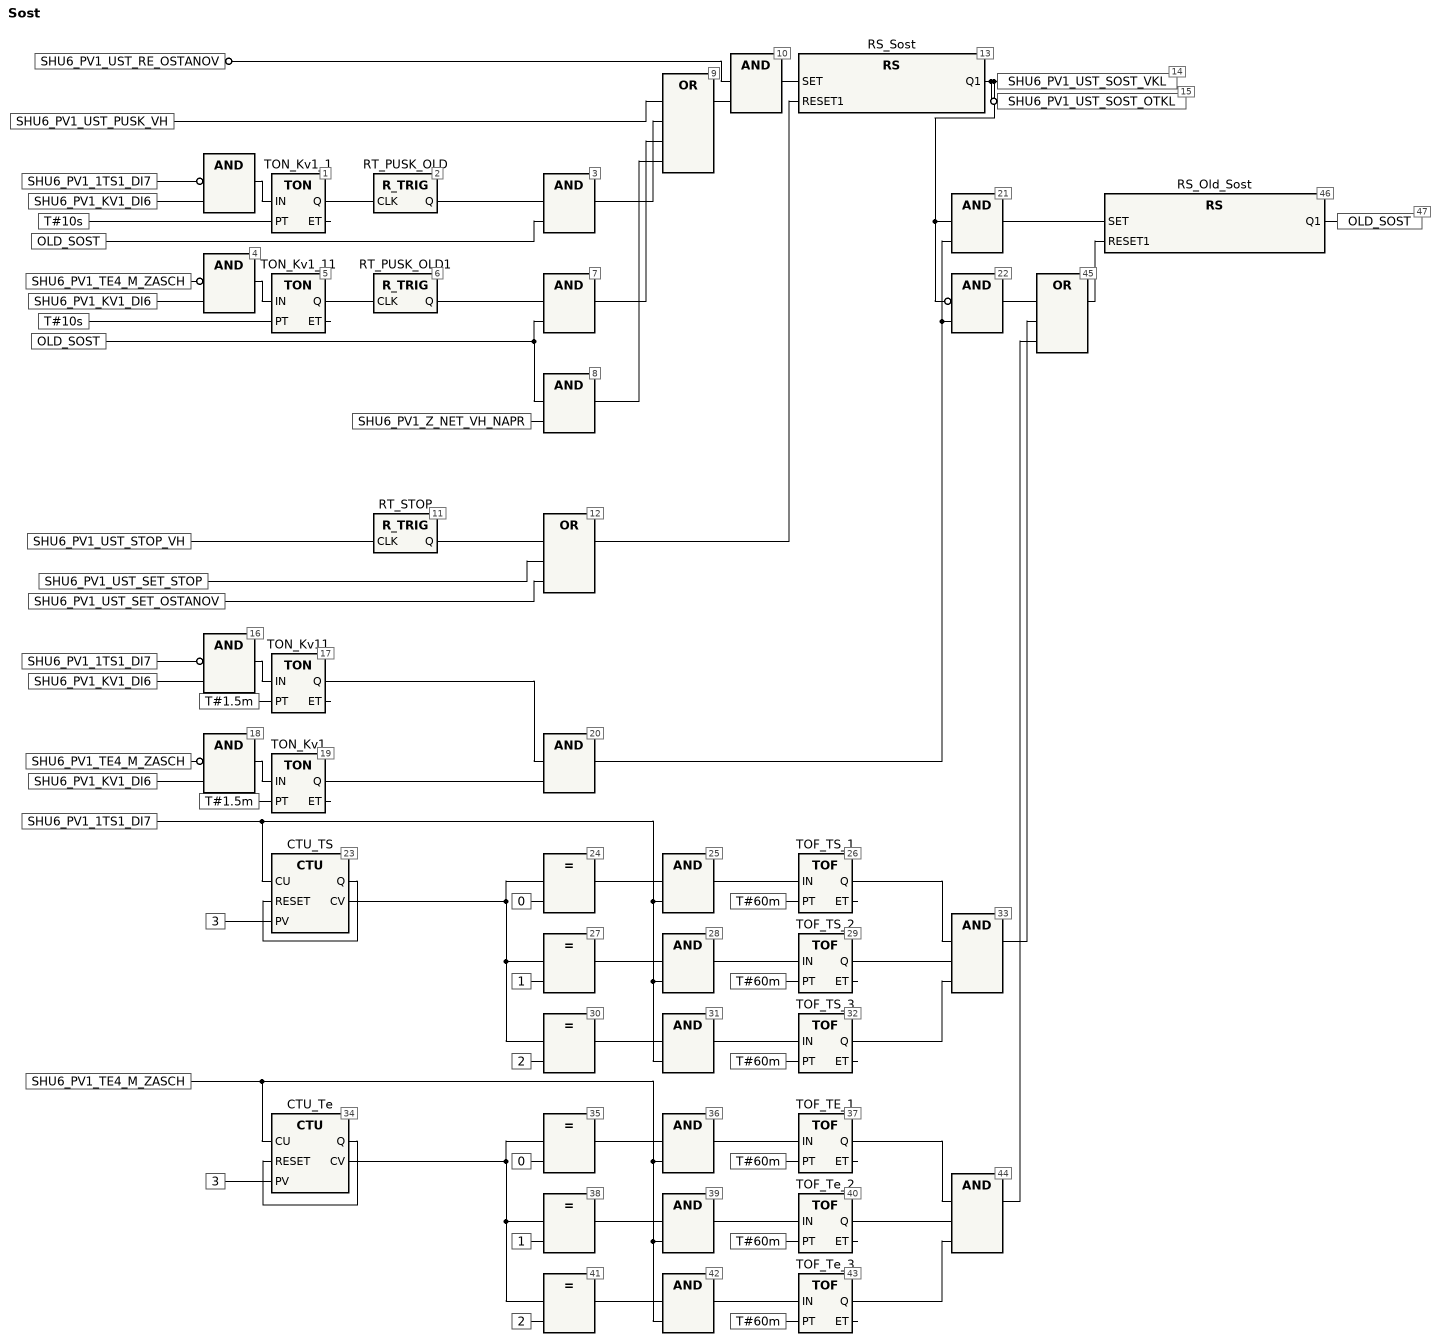
_CFC_ (* Continuous Function Chart, elements in execution order *)
#0 AND(NOT SHU6_PV1_1TS1_DI7, SHU6_PV1_KV1_DI6)
#1 TON_Kv1_1:TON(IN: #0, PT: T#10s)
#2 RT_PUSK_OLD:R_TRIG(CLK: #1.Q)
#3 AND(#2.Q, OLD_SOST)
#4 AND(NOT SHU6_PV1_TE4_M_ZASCH, SHU6_PV1_KV1_DI6)
#5 TON_Kv1_11:TON(IN: #4, PT: T#10s)
#6 RT_PUSK_OLD1:R_TRIG(CLK: #5.Q)
#7 AND(#6.Q, OLD_SOST)
#8 AND(OLD_SOST, SHU6_PV1_Z_NET_VH_NAPR)
#9 OR(SHU6_PV1_UST_PUSK_VH, #3, #7, #8)
#10 AND(NOT SHU6_PV1_UST_RE_OSTANOV, #9)
#11 RT_STOP:R_TRIG(CLK: SHU6_PV1_UST_STOP_VH)
#12 OR(#11.Q, SHU6_PV1_UST_SET_STOP, SHU6_PV1_UST_SET_OSTANOV)
#13 RS_Sost:RS(SET: #10, RESET1: #12)
#14 SHU6_PV1_UST_SOST_VKL <= #13.Q1
#15 SHU6_PV1_UST_SOST_OTKL <= NOT #13.Q1
#16 AND(NOT SHU6_PV1_1TS1_DI7, SHU6_PV1_KV1_DI6)
#17 TON_Kv11:TON(IN: #16, PT: T#1.5m)
#18 AND(NOT SHU6_PV1_TE4_M_ZASCH, SHU6_PV1_KV1_DI6)
#19 TON_Kv1:TON(IN: #18, PT: T#1.5m)
#20 AND(#17.Q, #19.Q)
#21 AND(#13.Q1, #20)
#22 AND(NOT #13.Q1, #20)
#23 CTU_TS:CTU(CU: SHU6_PV1_1TS1_DI7, RESET: #23.Q, PV: 3)
#24 =(#23.CV, 0)
#25 AND(#24, SHU6_PV1_1TS1_DI7)
#26 TOF_TS_1:TOF(IN: #25, PT: T#60m)
#27 =(#23.CV, 1)
#28 AND(#27, SHU6_PV1_1TS1_DI7)
#29 TOF_TS_2:TOF(IN: #28, PT: T#60m)
#30 =(#23.CV, 2)
#31 AND(#30, SHU6_PV1_1TS1_DI7)
#32 TOF_TS_3:TOF(IN: #31, PT: T#60m)
#33 AND(#26.Q, #29.Q, #32.Q)
#34 CTU_Te:CTU(CU: SHU6_PV1_TE4_M_ZASCH, RESET: #34.Q, PV: 3)
#35 =(#34.CV, 0)
#36 AND(#35, SHU6_PV1_TE4_M_ZASCH)
#37 TOF_TE_1:TOF(IN: #36, PT: T#60m)
#38 =(#34.CV, 1)
#39 AND(#38, SHU6_PV1_TE4_M_ZASCH)
#40 TOF_Te_2:TOF(IN: #39, PT: T#60m)
#41 =(#34.CV, 2)
#42 AND(#41, SHU6_PV1_TE4_M_ZASCH)
#43 TOF_Te_3:TOF(IN: #42, PT: T#60m)
#44 AND(#37.Q, #40.Q, #43.Q)
#45 OR(#22, #33, #44)
#46 RS_Old_Sost:RS(SET: #21, RESET1: #45)
#47 OLD_SOST <= #46.Q1
_END_CFC_
END_PROGRAM

(* POU Regim/Stop, CFC *)
PROGRAM Stop
VAR
	FT_Ostanov: F_TRIG;
	sr_stop: SR;
	TOF_Progrev: TOF;
END_VAR
VAR (* helpers for the ST form of the networks *)
	_t19 : BOOL;
END_VAR
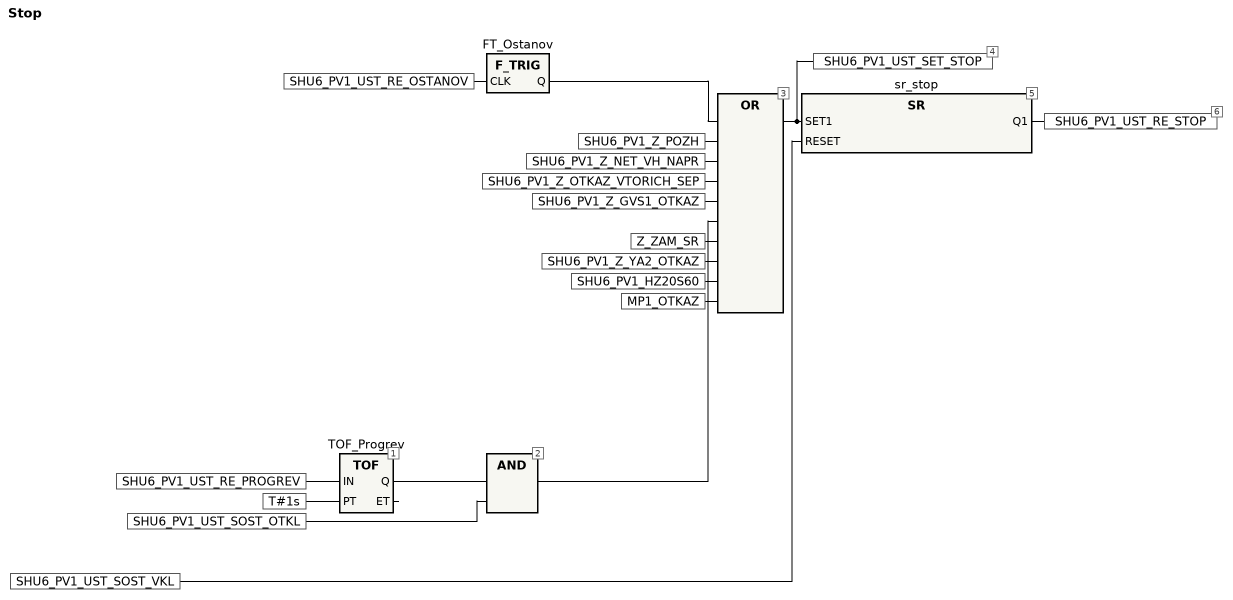
